Staubli VAL3: mergeVectors.pgx

public program mergeVectors(num& x_nInput_1[], num& x_nInput_2[], num& x_nResult[])
  local num l_nLength[2]
  local num l_nElement
begin

  l_nLength[0] = size(x_nInput_1)
  l_nLength[1] = size(x_nInput_2)
  resize(x_nResult,1,1)
  x_nResult[0] = 0
  resize(x_nResult,1,l_nLength[0]+l_nLength[1])

  // combine the two inputs
  for l_nElement = 0 to size(x_nResult)-1
    if l_nElement < l_nLength[0]
      x_nResult[l_nElement] = x_nInput_1[l_nElement]
    else
      x_nResult[l_nElement] = x_nInput_2[l_nElement-l_nLength[0]]
    endIf

  endFor

end
